TYPE T_PackedFb : FB_Packed; END_TYPE

(* stored: Version 1.1.0.1
   DUT T_PackedFb: Id {ad4d2d93-9a47-4003-8ac2-35dc8b8c555b} *)
